REGION Network 25: Super User
   RUNG wire#powerrail
      Contact( "Area02".AreaInterface.Man )
      Coil( "A02_HMI".Area02.SuperUser.SgnMan )
   END_RUNG
   RUNG wire#powerrail
      Contact( "Area02".AreaInterface.Aut )
      Coil( "A02_HMI".Area02.SuperUser.SgnAut )
   END_RUNG
   RUNG wire#powerrail
      Contact( "A02_HMI".Area02.SuperUser.PbReset )
      Coil( "A02_HMI".Area02.SuperUser.SgnReset )
   END_RUNG
   RUNG wire#powerrail
      Contact( "Area02".AreaInterface.Cycle )
      Coil( "A02_HMI".Area02.SuperUser.SgnStart )
   END_RUNG
   RUNG wire#powerrail
      { S7_Templates := "SrcType := Int" } GT_Contact(in1 := "A02_HMI".Area02.Status.WarningsNumber, in2 := 0)
      Coil( "A02_HMI".Area02.SuperUser.SgnWngPresence )
   END_RUNG
   RUNG wire#powerrail
      { S7_Templates := "SrcType := Int" } GT_Contact(in1 := "A02_HMI".Area02.Status.AlarmsNumber, in2 := 0)
      Coil( "A02_HMI".Area02.SuperUser.SgnAlrPresence )
   END_RUNG
   RUNG wire#powerrail
      Contact( false )
      Coil( "A02_HMI".Area02.SuperUser.SgnMessagePresence )
   END_RUNG
   RUNG wire#powerrail
      I_Contact( "Area02".AreaInterface.StopInPhase )
      I_Contact( "Area02".AreaInterface.StopProgrammed )
      Not()
      Coil( "A02_HMI".Area02.SuperUser.SgnStop )
   END_RUNG
   // the same network as SCL:
   "A02_HMI".Area02.SuperUser.SgnMan := "Area02".AreaInterface.Man;
   "A02_HMI".Area02.SuperUser.SgnAut := "Area02".AreaInterface.Aut;
   "A02_HMI".Area02.SuperUser.SgnReset := "A02_HMI".Area02.SuperUser.PbReset;
   "A02_HMI".Area02.SuperUser.SgnStart := "Area02".AreaInterface.Cycle;
   "A02_HMI".Area02.SuperUser.SgnWngPresence := "A02_HMI".Area02.Status.WarningsNumber > 0;
   "A02_HMI".Area02.SuperUser.SgnAlrPresence := "A02_HMI".Area02.Status.AlarmsNumber > 0;
   "A02_HMI".Area02.SuperUser.SgnMessagePresence := false;
   "A02_HMI".Area02.SuperUser.SgnStop := NOT (NOT "Area02".AreaInterface.StopInPhase AND NOT "Area02".AreaInterface.StopProgrammed);
END_REGION

REGION Network 26 (SCL): <<< MACHINES AREA 02 >>>
   "A02_HMI_CALL"();

   "A02_ButtonSafe_CALL"();

   "RollformingMng_CALL"();

   "PostPunchingMatCounter_CALL"();

   "MwFakCalc_CALL"();

   "WeldReg_CALL"();

   "Area02_HU_CALL"();

   "A0201_Profilatrice_RegolazioneFormato_OB1_CALL"();

   "PitTable1_CALL"();

   "Rollformer_CALL"();

   "RollfomrerLubr_CALL"();

   "FlyingCarriage_CALL"();

   "CarriageLub_CALL"();

   "FinalCut_CALL"();

   "FinalCutLub_CALL"();

   "AccRollConveyor_CALL"();

   "A02_TrkManager_CALL"();
END_REGION

REGION Network 27: >
END_REGION

REGION Network 28: Area ITF Orchestrator
   RUNG wire#powerrail
      "Area02_ITF"()
   END_RUNG
   // the same network as SCL:
   "Area02_ITF"();
END_REGION

REGION Network 29: >
END_REGION

REGION Network 30: >
END_REGION
END_FUNCTION
